# B&R Automation Studio project trialproject2
Automation Studio 4.5.2.102

## Configuration labBR

### Task classes (Cpu.sw)
```
Cyclic#1 (cycle 2000 us, tolerance 0 us):
  ncsdcctrl <- ncsdcctrl.prg
Cyclic#3:
  Program_LE <- Program_LED.prg
Cyclic#4:
  drive_cont <- drive_control.prg
DataObjects: Acp10sys
NcDataObjects: acp10etxen <- acp10etxen.dob, gAxis01a <- gAxis01obj.gAxis01a.dob, gAxis01i <- gAxis01obj.gAxis01i.dob
VcDataObjects: Visu <- Visu.dob
Binaries: vcpdsw, udbdef, vcrt, vcctext, vcpfmtcx, Visu03, vcfile, vcgclass, arial, vcdsint, vcmgr, vcdsloc, vcfntttf, Visu02, vccovl, vcshared, arialbd, vcalarm, vcptelo, vccdt, vccline, vcpdpp30, vccbtn, Visu01, vcbclass, vcpfpp30, vctcal, TCData, vcctrend, vccgauge, iomap, asfw, Role, ashwac, sysconf, ashwd, User, arconfig, acp10cfg, Acp10map
Libraries: Acp10man, Acp10par, NcGlobal, Acp10sdc, AsBrStr, Acp10_MC, brsystem, sys_lib, runtime, vcresman, asieccon, fileio, astime, dataobj, powerlnk, Library
```

### Hardware
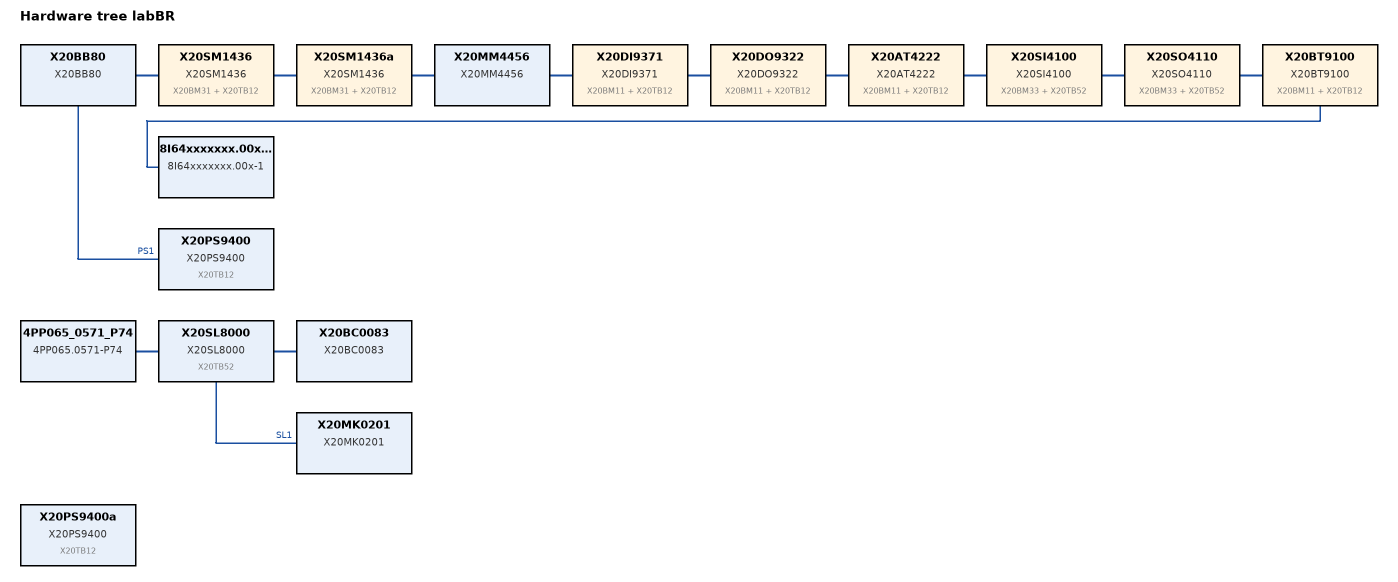
```
4PP065_0571_P74 : 4PP065.0571-P74 v1.1.2.0
  Connector IF5:
    ActivateDevice = 1
    Mode = Manual
    InternetAddress = 10.0.1.10
    SubnetMask = 255.255.255.0
  ConfigurationID = labBR
  TimerDeviceType = EPLX2X
  TimerDevice = 4PP065_0571_P74.IF4
  TaskClassIdleTime = 2000
  Cyclic1Duration = 2000
  Cyclic1Tolerance = 0
  Cyclic1Output = 1
  VcObjectName = Visu
8I64xxxxxxx.00x-1 : 8I64xxxxxxx.00x-1 v2.1.2.0  [X2X1 -> X20BT9100.X2X1 [Cable Type=X2XCable, Length=10, Version=1.0.0.2]]
  packedETAD = packed
  packedCMDD = packed
X20AT4222 : X20AT4222 v1.2.3.0  [SS1 -> X20TB12f.SS; SL -> X20BM11b.SL1]
X20BB80 : X20BB80 v1.0.2.0
X20BC0083 : X20BC0083 v2.9.0.0  [PLK1 -> X20SL8000.PLK2 [Cable Type=PowerlinkCable, Length=10, Version=1.0.0.2]; SL -> X20BB80.SL1]
X20BM11 : X20BM11 v1.0.0.1  [X2X1 -> X20MM4456.X2X2]
X20BM11a : X20BM11 v1.0.0.1  [X2X1 -> X20BM11.X2X2]
X20BM11b : X20BM11 v1.0.0.1  [X2X1 -> X20BM11a.X2X2]
X20BM11c : X20BM11 v1.0.0.1  [X2X1 -> X20BM33a.X2X2]
X20BM31 : X20BM31 v1.0.0.1  [X2X1 -> X20BB80.IF1]
X20BM31a : X20BM31 v1.0.0.1  [X2X1 -> X20BM31.X2X2]
X20BM33 : X20BM33 v1.0.0.4  [X2X1 -> X20BM11b.X2X2]
X20BM33a : X20BM33 v1.0.0.4  [X2X1 -> X20BM33.X2X2]
X20BT9100 : X20BT9100 v1.0.3.0  [SS1 -> X20TB12g.SS; SL -> X20BM11c.SL1]
X20DI9371 : X20DI9371 v1.0.2.0  [SS1 -> X20TB12d.SS; SL -> X20BM11.SL1]
X20DO9322 : X20DO9322 v1.0.3.0  [SS1 -> X20TB12e.SS; SL -> X20BM11a.SL1]
X20MK0201 : X20MK0201 v1.0.0.0  [SL -> X20SL8000.SL1]
X20MM4456 : X20MM4456 v1.1.5.0  [X2X1 -> X20BM31a.X2X2]
X20PS9400 : X20PS9400 v1.8.0.0  [SS1 -> X20TB12.SS; PS -> X20BB80.PS1]
X20PS9400a : X20PS9400 v1.8.0.0  [SS1 -> X20TB12a.SS]
X20SI4100 : X20SI4100 v1.10.1.1  [SS1 -> X20TB52a.SS; SL -> X20BM33.SL1]
X20SL8000 : X20SL8000 v1.6.5.2  [PLK1 -> 4PP065_0571_P74.IF4 [Cable Type=PowerlinkCable, Length=10, Version=1.0.0.2]; PLK2 -> X20BC0083.PLK1 [Cable Type=PowerlinkCable, Length=10, Version=1.0.0.2]; SS1 -> X20TB52.SS]
  SafeProject = SafeLOGIC-1
X20SM1436 : X20SM1436 v2.2.0.0  [SS1 -> X20TB12b.SS; SL -> X20BM31.SL1]
  MotionTP = Acp10Arnc0
X20SM1436a : X20SM1436 v2.2.0.0  [SS1 -> X20TB12c.SS; SL -> X20BM31a.SL1]
  MotionTP = Acp10Arnc0
X20SO4110 : X20SO4110 v1.10.1.1  [SS1 -> X20TB52b.SS; SL -> X20BM33a.SL1]
  SafeModuleID = 3
X20TB12 : X20TB12 v1.0.0.0
X20TB12a : X20TB12 v1.0.0.0
X20TB12b : X20TB12 v1.0.0.0
X20TB12c : X20TB12 v1.0.0.0
X20TB12d : X20TB12 v1.0.0.0
X20TB12e : X20TB12 v1.0.0.0
X20TB12f : X20TB12 v1.0.0.0
X20TB12g : X20TB12 v1.0.0.0
X20TB52 : X20TB52 v1.0.0.1
X20TB52a : X20TB52 v1.0.0.1
X20TB52b : X20TB52 v1.0.0.1
```

### IoMap.iom - 4PP065_0571_P74/IoMap.iom
```iecst
VAR_CONFIG
	Cyclic#1.gAxis01_DrvIf.iLifeCnt AT %IB."8I64xxxxxxx.00x-1".SDC_LifeCnt;
	Cyclic#1.gAxis01_DrvIf.iDrvOK AT %IX."8I64xxxxxxx.00x-1".ETAD_Input_Bool_02;
	Cyclic#1.gAxis01_DrvIf.oSetTime AT %QW."8I64xxxxxxx.00x-1".SDC_SetTime;
	Cyclic#1.::speed AT %QW."8I64xxxxxxx.00x-1".LFRD_Output;
	Cyclic#1.gAxis01_DiDoIf.iLifeCntDriveReady AT %IB."8I64xxxxxxx.00x-1".SDC_LifeCnt;
	Cyclic#1.gAxis01_DiDoIf.iLifeCntDriveEnable AT %IB."8I64xxxxxxx.00x-1".SDC_LifeCnt;
	Cyclic#1.gAxis01_DiDoIf.oDriveEnable AT %QX."8I64xxxxxxx.00x-1".CMDD_Output_Bool_00;
	Cyclic#1.gAxis01_ModuleOk AT %QX."8I64xxxxxxx.00x-1".CMDD_Output_Bool_01;
	Cyclic#1.gAxis01_ModuleOk AT %QX."8I64xxxxxxx.00x-1".CMDD_Output_Bool_02;
	Cyclic#1.gAxis01_ModuleOk AT %IX."8I64xxxxxxx.00x-1".ModuleOk;
	Cyclic#1.gAxis01_DiDoIf.oDriveEnable AT %QX."8I64xxxxxxx.00x-1".CMDD_Output_Bool_03;
	Cyclic#1.gAxis01_DiDoIf.iDriveReady AT %IX."8I64xxxxxxx.00x-1".ETAD_Input_Bool_02;
	::LED[0] AT %QX."X20DO9322".DigitalOutput02;
	::LED[1] AT %QX."X20DO9322".DigitalOutput03;
	::LED[2] AT %QX."X20DO9322".DigitalOutput04;
	::LED[3] AT %QX."X20DO9322".DigitalOutput05;
	::EVRID.STATE AT %IW."8I64xxxxxxx.00x-1".ETAD_Input;
	::EVRID.CMD AT %QW."8I64xxxxxxx.00x-1".CMDD_Output;
	::EVRID.real_speed AT %IW."8I64xxxxxxx.00x-1".RFRD_Input;
END_VAR
```

## Logical view

Binary libraries used (declarations not repeated): operator, Acp10man, runtime, astime, AsIecCon, Acp10par, NcGlobal, Acp10sdc, AsBrStr, Acp10_MC, brsystem, sys_lib

### Global.var - Global variables
```iecst
VAR
	speed : INT;
	gAxis01 : ACP10AXIS_typ;
	gAxis01_HW : SdcHwCfg_typ := (0);
	gAxis01_DrvIf : SdcDrvIf16_typ := (0);
	gAxis01_DiDoIf : SdcDiDoIf_typ := (0);
	gAxis01_ModuleOk : BOOL := 0;
	LED : ARRAY[0..3] OF BOOL := [4(0)];
	button1 : BOOL := FALSE;
	button2 : BOOL := FALSE;
	button3 : BOOL := FALSE;
	button4 : BOOL := FALSE;
	button5 : BOOL := FALSE;
	counter : USINT := 0;
	EVRID : DRIVE;
END_VAR
```

### Package Logical/Libraries - Global libraries

### Library Logical/Libraries/Library (ANSIC)

#### Constants.var
```iecst
VAR CONSTANT
	CMD_SWITCHED_ON : UINT := 7;
	CMD_DISABLED_VOLTAGE : UINT := 0;
	CMD_ENABLED : UINT := 15;
	CMD_SHUTDOWN : UINT := 6;
	STATE_DISABLED : UINT := 64;
	STATE_READY : UINT := 33;
	STATE_SWITCHED_ON : USINT := 35;
END_VAR
```

#### Library.fun
```iecst
{REDUND_ERROR} FUNCTION_BLOCK DRIVE (*TODO: Add your comment here*) (*$GROUP=User,$CAT=User,$GROUPICON=User.png,$CATICON=User.png*)
	VAR_INPUT
		ENABLE : BOOL;
	END_VAR
	VAR_OUTPUT
		real_speed : INT;
	END_VAR
	VAR_INPUT
		STATE : UINT;
	END_VAR
	VAR_OUTPUT
		CMD : UINT;
	END_VAR
END_FUNCTION_BLOCK
```

#### DRIVE.c
```c
#include <bur/plctypes.h>
#ifdef __cplusplus
	extern "C"
	{
#endif
	#include "Library.h"
#ifdef __cplusplus
	};
#endif
/* TODO: Add your comment here */
void DRIVE(struct DRIVE* inst)
{
	UINT mask=inst->STATE & 0x6f;
	if(!inst->ENABLE){
		inst->CMD = CMD_SHUTDOWN;
	}
	else{
		switch (mask)
		{
			case STATE_DISABLED:

				inst->CMD=CMD_SHUTDOWN;
				break;
			case STATE_READY:

				inst->CMD=CMD_ENABLED;
				break;
			case STATE_SWITCHED_ON:

				inst->CMD=CMD_SWITCHED_ON;
				break;
		}
	}
}
```

- Visualisation Logical/Visu (not shown)

### Program Logical/Program_LED (ANSIC)

#### Main.c
```c
#include <bur/plctypes.h>

#ifdef _DEFAULT_INCLUDES
	#include <AsDefault.h>
#endif

void _INIT ProgramInit(void)
{

}

void _CYCLIC ProgramCyclic(void)
{
	if (button5 == 1){
		if(counter%2 == 0){
			LED[0]=!LED[0];
		}
		if(counter%4 == 0){
			LED[1]=!LED[1];
		}
		if(counter%8 == 0){
			LED[2]=!LED[2];
		}
		if(counter%16 == 0){
			LED[3]=!LED[3];
		}
		counter++;

	}
	else{
		LED[0] = button1;
		LED[1] = button2;
		LED[2] = button3;
		LED[3] = button4;
	}
}
void _EXIT ProgramExit(void)
{

}
```

### Program Logical/drive_control (ANSIC)

#### Main.c
```c
#include <bur/plctypes.h>

#ifdef _DEFAULT_INCLUDES
	#include <AsDefault.h>
#endif

void _INIT ProgramInit(void)
{
	speed = 0;
	EVRID.ENABLE = 1;
}

void _CYCLIC ProgramCyclic(void)
{
	DRIVE(&EVRID);
}

void _EXIT ProgramExit(void)
{

}
```

Listed in the project but not available here: Logical/Global.typ, Logical/acp10etxen, Logical/ncsdcctrl, Logical/gAxis01obj
